Universal Robots PolyScope program: Project1pick4.urp

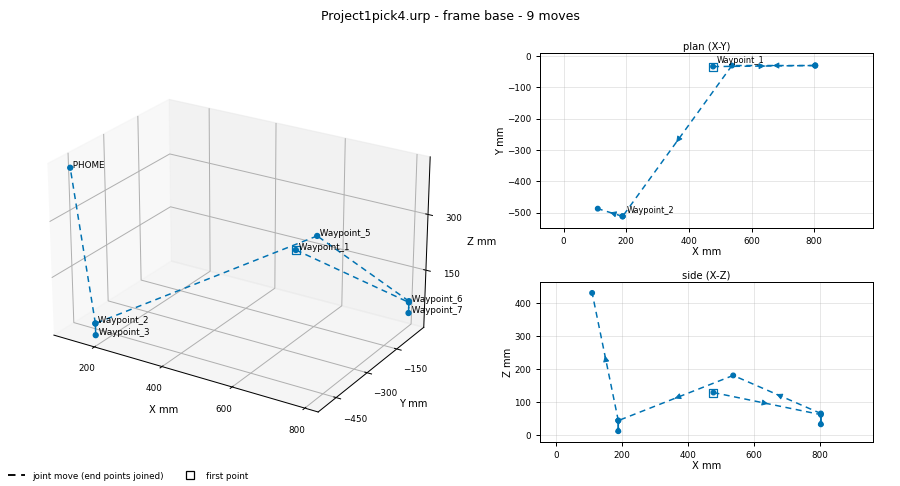
[picture p0: tool path of Project1pick4.urp in frame base, 9 of 9 moves have a stored position in this frame; points joined in program order, loops and branches not executed]
Program Project1pick4 (installation=admin directory=/programs/TUES_530PM createdIn=3.15.8.106339 lastSavedIn=3.15.8.106339 robotSerialNumber=2015350926)
Calibrated DH parameters: a=[0, -0.425, -0.39225, 0, 0, 0]; d=[0.089159, 0, 0, 0.10915, 0.09465, 0.0823]; alpha=[1.570796, 0, 0, 1.570796, -1.570796, 0]; deltaTheta=[0, 0, 0, 0, 0, 0]
Robot Program (runOnlyOnce=true)
  MoveJ speed 60 deg/s, acceleration 80 deg/s^2 (useActiveTCP=true)
    Waypoint Waypoint_1: TCP in base x=477.218 y=-33.357 z=129.572 mm, rx=2.2261 ry=-2.212 rz=0.0055 rad; joints [162.86, -75.572, 123.035, -137.55, -90.266, -17.505] deg
    Waypoint Waypoint_6: TCP in base x=803.264 y=-30.051 z=62.587 mm, rx=2.2261 ry=-2.212 rz=0.0057 rad; joints [170.082, -33.741, 61.128, -117.446, -90.277, -10.281] deg
    Waypoint Waypoint_7: TCP in base x=803.244 y=-30.061 z=33.168 mm, rx=2.226 ry=-2.2118 rz=0.0054 rad; joints [170.081, -31.572, 61.598, -120.071, -90.28, -10.283] deg
    Wait Sleep waitTime=0.5
    Set DigitalOutput pin=digital_out[0]; digitalValue=1
    Wait Sleep waitTime=0.5
    Waypoint Waypoint_4: TCP in base x=803.272 y=-30.057 z=66.011 mm, rx=2.226 ry=-2.2119 rz=0.0055 rad; joints [170.082, -33.98, 61.044, -117.115, -90.281, -10.283] deg
    Waypoint Waypoint_5: TCP in base x=537.259 y=-30.095 z=181.531 mm, rx=2.2259 ry=-2.2118 rz=0.0054 rad; joints [165.134, -73.968, 110.575, -126.676, -90.279, -15.23] deg
    Waypoint Waypoint_2: TCP in base x=188.485 y=-511.481 z=44.451 mm, rx=2.2261 ry=-2.2117 rz=0.0056 rad; joints [98.685, -58.69, 114.899, -146.495, -90.041, -81.687] deg
    Waypoint Waypoint_3: TCP in base x=188.431 y=-511.439 z=12.275 mm, rx=2.226 ry=-2.2118 rz=0.0056 rad; joints [98.68, -54.617, 115.165, -150.832, -90.043, -81.687] deg
    Wait Sleep waitTime=0.5
    Set DigitalOutput pin=digital_out[0]; digitalValue=0
    Wait Sleep waitTime=0.5
    Waypoint Waypoint_2: TCP in base x=188.485 y=-511.481 z=44.451 mm, rx=2.2261 ry=-2.2117 rz=0.0056 rad; joints [98.685, -58.69, 114.899, -146.495, -90.041, -81.687] deg
    Waypoint PHOME: TCP in base x=109.127 y=-486.917 z=431.88 mm, rx=0.0001 ry=3.1416 rz=-0.0002 rad; joints [89.997, -90, 89.999, -90.006, -89.998, 0.001] deg
